// TIA Portal V15.1 export
// export: Created 2024-06-21T08:41:13.6587358Z, ExportSetting WithDefaults, DisplayName Totally Integrated Automation Portal, DisplayVersion V15.1 Update 5, DisplayName TIA Portal Openness, DisplayVersion V15.1 Update 5, DisplayName SINAMICS Startdrive Advanced, DisplayVersion V15.1, DisplayName G130, G150, S120, S150, SINAMICS MV, S210, DisplayVersion V15.1, DisplayName G110M, G120, G120C, G120D, G120P, DisplayVersion V15.1, DisplayName STEP 7 Professional, DisplayVersion V15.1 Update 5, DisplayName STEP 7 Safety, DisplayVersion V15.1, DisplayName WinCC Professional, DisplayVersion V15.1 Update 5, DisplayName SIMATIC Visualization Architect, DisplayVersion V15.1
FUNCTION_BLOCK "LGBLightCurtain"   // FB6634, FBD
TITLE = LGBLightCurtain
{ S7_Optimized_Access := 'FALSE' }
VERSION : 0.1
// ============================================================================
// This module is generates an alarm regarding a light curtain. The module manages also the bypass key and the pollution alarm.
// The light curtain alarm is reset by means of the AlarmResetPB signal.
// 
// This module generates also a word containing all necessary information for HMI 
// Icon animation, and a word with all information for HMI safety module diagnostic screen. 
// ============================================================================
// stored: AutoNumber false, IsIECCheckEnabled false, SetENOAutomatically False, UDAEnableTagReadback false
   VAR_INPUT
      I_LightCurtain { ExternalAccessible := 'False'; ExternalVisible := 'False'; ExternalWritable := 'False'} : Bool;   // Input safety (normally closed) / Input safety alarm (normally closed)
      I_Polluted { ExternalAccessible := 'False'; ExternalVisible := 'False'; ExternalWritable := 'False'} : Bool;   // Light curtain is polluted / Input safety alarm (normally closed)
      I_MutingAlarm { ExternalAccessible := 'False'; ExternalVisible := 'False'; ExternalWritable := 'False'} : Bool;   // Muting alarm from safety FB "MUT_P"
      I_OkToReset { ExternalAccessible := 'False'; ExternalVisible := 'False'; ExternalWritable := 'False'} : Bool;   // Ok to Reset Light curtain
      I_BypassKey { ExternalAccessible := 'False'; ExternalVisible := 'False'; ExternalWritable := 'False'} : Bool;   // Light curtain override key is turned / Input safety alarm (normally closed)
      I_AlarmClassLightCurtain { ExternalAccessible := 'False'; ExternalVisible := 'False'; ExternalWritable := 'False'} : Char;   // Alarm class -> A - B - C - D or E
      I_AlarmClassMuting { ExternalAccessible := 'False'; ExternalVisible := 'False'; ExternalWritable := 'False'} : Char;   // Alarm class -> A - B - C - D or E
      I_EnableAlarm { ExternalAccessible := 'False'; ExternalVisible := 'False'; ExternalWritable := 'False'} : Bool := TRUE;   // Enable alarm from upper level
      I_AlarmResetPB { ExternalAccessible := 'False'; ExternalVisible := 'False'; ExternalWritable := 'False'} : Bool;   // Alarm reset pushbutton is activated
      I_ResetAlarmPolluted { ExternalAccessible := 'False'; ExternalVisible := 'False'; ExternalWritable := 'False'} : Bool;   // Reset polluted alarm / Alarm reset pushbutton is activated
      I_SafetyCard_PASS_OUT { ExternalAccessible := 'False'; ExternalVisible := 'False'; ExternalWritable := 'False'} : Bool;   // Automatically generated DB from F-Modul (F-Peripherie DB)
      I_SafetyCard_ACK_REQ { ExternalAccessible := 'False'; ExternalVisible := 'False'; ExternalWritable := 'False'} : Bool;   // Automatically generated DB from F-Modul (F-Peripherie DB)
      I_SafetyCard_DIAG { ExternalAccessible := 'False'; ExternalVisible := 'False'; ExternalWritable := 'False'} : Byte;   // Automatically generated DB from F-Modul (F-Peripherie DB)
      I_SafetyCardHWSub { ExternalAccessible := 'False'; ExternalVisible := 'False'; ExternalWritable := 'False'} : HW_SUBMODULE;   // Safety I/O connection hardware
      I_ChannelNr { ExternalAccessible := 'False'; ExternalVisible := 'False'; ExternalWritable := 'False'} : Int;   // Used Channel Nr (Value : 0, 1, 2, 3)
      C_DisableQBadCh { ExternalAccessible := 'False'; ExternalVisible := 'False'; ExternalWritable := 'False'} : Bool;   // Passivation Channel (QbadCh1) / Disable QBad Channel
      C_DisablePollutedAlarm { ExternalAccessible := 'False'; ExternalVisible := 'False'; ExternalWritable := 'False'} : Bool;   // Disable Polluted Alarm
   END_VAR
   VAR_OUTPUT
      O_AlarmABCondition { ExternalAccessible := 'False'; ExternalVisible := 'False'; ExternalWritable := 'False'} : Bool;   // Alarm AB condition
      O_AlarmA { ExternalAccessible := 'False'; ExternalVisible := 'False'; ExternalWritable := 'False'} : Bool;   // Alarm A
      O_AlarmB { ExternalAccessible := 'False'; ExternalVisible := 'False'; ExternalWritable := 'False'} : Bool;   // Alarm B
      O_AlarmC { ExternalAccessible := 'False'; ExternalVisible := 'False'; ExternalWritable := 'False'} : Bool;   // Alarm C
      O_AlarmD { ExternalAccessible := 'False'; ExternalVisible := 'False'; ExternalWritable := 'False'} : Bool;   // Alarm D
      H_IAnim { ExternalAccessible := 'False'; ExternalVisible := 'False'; ExternalWritable := 'False'} : DWord;   // Icon Animation
      H_AlarmWord { ExternalAccessible := 'False'; ExternalVisible := 'False'; ExternalWritable := 'False'} : DWord;   // Alarm Word
   END_VAR
   VAR DB_SPECIFIC
      H_Out : Struct   // HMI
         Anim : Word;   // HMI Animation of the object
         DBnr : Int;   // HMI Animation DB number
      END_STRUCT;
      AlarmClassLightCurtain_A { ExternalAccessible := 'False'; ExternalVisible := 'False'; ExternalWritable := 'False'} : Bool;   // The alarm is from alarm class A / The alarm is from alarm Light Curtain class A
      AlarmClassLightCurtain_B { ExternalAccessible := 'False'; ExternalVisible := 'False'; ExternalWritable := 'False'} : Bool;   // The alarm is from alarm class B / The alarm is from alarm Light Curtain class B
      AlarmClassLightCurtain_C { ExternalAccessible := 'False'; ExternalVisible := 'False'; ExternalWritable := 'False'} : Bool;   // The alarm is from alarm class C / The alarm is from alarm Light Curtain class C
      AlarmClassLightCurtain_D { ExternalAccessible := 'False'; ExternalVisible := 'False'; ExternalWritable := 'False'} : Bool;   // The alarm is from alarm class D / The alarm is from alarm Light Curtain class D
      AlarmClassMuting_A { ExternalAccessible := 'False'; ExternalVisible := 'False'; ExternalWritable := 'False'} : Bool;   // The alarm is from alarm class A / The alarm is from alarm Muting class A
      AlarmClassMuting_B { ExternalAccessible := 'False'; ExternalVisible := 'False'; ExternalWritable := 'False'} : Bool;   // The alarm is from alarm class B / The alarm is from alarm Muting class B
      AlarmClassMuting_C { ExternalAccessible := 'False'; ExternalVisible := 'False'; ExternalWritable := 'False'} : Bool;   // The alarm is from alarm class C / The alarm is from alarm Muting class C
      AlarmClassMuting_D { ExternalAccessible := 'False'; ExternalVisible := 'False'; ExternalWritable := 'False'} : Bool;   // The alarm is from alarm class D / The alarm is from alarm Muting class D
      Alarm { ExternalAccessible := 'False'; ExternalVisible := 'False'; ExternalWritable := 'False'} : Bool;   // Alarm
      AA_LightCurtainAlarm { ExternalAccessible := 'False'; ExternalVisible := 'False'; ExternalWritable := 'False'} : Bool;   // Alarm of the light curtain / Alarm
      AB_LightCurtainAlarm { ExternalAccessible := 'False'; ExternalVisible := 'False'; ExternalWritable := 'False'} : Bool;   // Alarm of the light curtain / Alarm
      AC_LightCurtainAlarm { ExternalAccessible := 'False'; ExternalVisible := 'False'; ExternalWritable := 'False'} : Bool;   // Alarm of the light curtain / Alarm
      AD_LightCurtainAlarm { ExternalAccessible := 'False'; ExternalVisible := 'False'; ExternalWritable := 'False'} : Bool;   // Alarm of the light curtain / Alarm
      AA_MutingAlarm { ExternalAccessible := 'False'; ExternalVisible := 'False'; ExternalWritable := 'False'} : Bool;   // Muting is not ok
      AB_MutingAlarm { ExternalAccessible := 'False'; ExternalVisible := 'False'; ExternalWritable := 'False'} : Bool;   // Muting is not ok
      AC_MutingAlarm { ExternalAccessible := 'False'; ExternalVisible := 'False'; ExternalWritable := 'False'} : Bool;   // Muting is not ok
      AD_MutingAlarm { ExternalAccessible := 'False'; ExternalVisible := 'False'; ExternalWritable := 'False'} : Bool;   // Muting is not ok
      AC_Polluted { ExternalAccessible := 'False'; ExternalVisible := 'False'; ExternalWritable := 'False'} : Bool;   // Light curtain is polluted / Alarm
      AC_Bypass { ExternalAccessible := 'False'; ExternalVisible := 'False'; ExternalWritable := 'False'} : Bool;   // Bypass key is activated / Alarm
      QbadCh1 { ExternalAccessible := 'False'; ExternalVisible := 'False'; ExternalWritable := 'False'} : Bool;   // Passivation first Channel
      Ack_Req { ExternalAccessible := 'False'; ExternalVisible := 'False'; ExternalWritable := 'False'} : Bool;   // Acknowledgement request
      Timeout_F_I_O { ExternalAccessible := 'False'; ExternalVisible := 'False'; ExternalWritable := 'False'} : Bool;   // Timeout detected by F-I/O
      ChannelFault_F_I_O { ExternalAccessible := 'False'; ExternalVisible := 'False'; ExternalWritable := 'False'} : Bool;   // F-I/O fault or channel fault detected by F-I/O
      CRCSeqError_F_I_O { ExternalAccessible := 'False'; ExternalVisible := 'False'; ExternalWritable := 'False'} : Bool;   // CRC error or sequence number error detected by F-I/O
      Timeout_F_Sys { ExternalAccessible := 'False'; ExternalVisible := 'False'; ExternalWritable := 'False'} : Bool;   // Timeout detected by F-System
      SeqError_F_Sys { ExternalAccessible := 'False'; ExternalVisible := 'False'; ExternalWritable := 'False'} : Bool;   // Sequence number error detected by F-system
      CRCError_F_Sys { ExternalAccessible := 'False'; ExternalVisible := 'False'; ExternalWritable := 'False'} : Bool;   // CRC error detected by F-system
      AlarmCond { ExternalAccessible := 'False'; ExternalVisible := 'False'; ExternalWritable := 'False'} : Bool;   // Alarm condition
      RetValueData { ExternalAccessible := 'False'; ExternalVisible := 'False'; ExternalWritable := 'False'} : Int;   // Status variable (SFC14)
      DBnr { ExternalAccessible := 'False'; ExternalVisible := 'False'; ExternalWritable := 'False'} : Int;   // HMI DB number
      AlarmABCondition { ExternalAccessible := 'False'; ExternalVisible := 'False'; ExternalWritable := 'False'} : Bool;   // Alarm AB Condition / Summation Alarm A
      AlarmA { ExternalAccessible := 'False'; ExternalVisible := 'False'; ExternalWritable := 'False'} : Bool;   // Summation Alarm A
      AlarmB { ExternalAccessible := 'False'; ExternalVisible := 'False'; ExternalWritable := 'False'} : Bool;   // Summation Alarm B
      AlarmC { ExternalAccessible := 'False'; ExternalVisible := 'False'; ExternalWritable := 'False'} : Bool;   // Summation Alarm C
      AlarmD { ExternalAccessible := 'False'; ExternalVisible := 'False'; ExternalWritable := 'False'} : Bool;   // Summation Alarm D
   END_VAR
   VAR_TEMP
      T_DataFromSafetyCard : Struct   // Temp structure : receive data's from Safety Card
         Byte0_Bit0_Spare : Bool;
         Byte0_Bit1_Spare : Bool;
         Byte0_Bit2_Spare : Bool;
         Byte0_Bit3_Spare : Bool;
         Byte0_Bit4_Spare : Bool;
         Byte0_Bit5_Spare : Bool;
         Byte0_Bit6_Spare : Bool;
         Byte0_Bit7_Spare : Bool;
         Byte1_Bit0_QBadCh0 : Bool;
         Byte1_Bit1_QBadCh1 : Bool;
         Byte1_Bit2_QBadCh2 : Bool;
         Byte1_Bit3_QBadCh3 : Bool;
         Byte1_Bit4_QBadCh4 : Bool;
         Byte1_Bit5_QBadCh5 : Bool;
         Byte1_Bit6_QBadCh6 : Bool;
         Byte1_Bit7_QBadCh7 : Bool;
         Byte2_bit0_Spare : Bool;
         Byte2_bit1_Spare : Bool;
         Byte2_bit2_Spare : Bool;
         Byte2_bit3_Spare : Bool;
         Byte2_bit4_Spare : Bool;
         Byte2_bit5_Spare : Bool;
         Byte2_bit6_Spare : Bool;
         Byte2_bit7_Spare : Bool;
         Byte3_Bit0_Spare : Bool;
         Byte3_Bit1_Spare : Bool;
         Byte3_Bit2_Spare : Bool;
         Byte3_Bit3_Spare : Bool;
         Byte3_Bit4_Spare : Bool;
         Byte3_Bit5_Spare : Bool;
         Byte3_Bit6_Spare : Bool;
         Byte3_Bit7_Spare : Bool;
         Byte4_bit0_Spare : Bool;
         Byte4_bit1_Spare : Bool;
         Byte4_bit2_Spare : Bool;
         Byte4_bit3_Spare : Bool;
         Byte4_bit4_Spare : Bool;
         Byte4_bit5_Spare : Bool;
         Byte4_bit6_Spare : Bool;
         Byte4_bit7_Spare : Bool;
         Byte5_bit0_Spare : Bool;
         Byte5_bit1_Spare : Bool;
         Byte5_bit2_Spare : Bool;
         Byte5_bit3_Spare : Bool;
         Byte5_bit4_Spare : Bool;
         Byte5_bit5_Spare : Bool;
         Byte5_bit6_Spare : Bool;
         Byte5_bit7_Spare : Bool;
      END_STRUCT;
   END_VAR
   VAR_TEMP   // added for the SCL form of the ladder/FBD networks
      _w1 : Bool;
   END_VAR
BEGIN

NETWORK
TITLE = **** 1 - Inputs **** DB number
// DB number
      L     DINO;
      T     #DBnr;

NETWORK
TITLE = **** 1 - Inputs **** Alarm class / **** 1 - Inputs **** Alarm class Light Curtain
// Alarm class
// Alarm class = D
      L     #I_AlarmClassLightCurtain;
      L     'D';
      ==I;
      =     #AlarmClassLightCurtain_D;

// Alarm class = C
      L     #I_AlarmClassLightCurtain;
      L     'C';
      ==I;
      =     #AlarmClassLightCurtain_C;

// Alarm class = B
      L     #I_AlarmClassLightCurtain;
      L     'B';
      ==I;
      =     #AlarmClassLightCurtain_B;

// Alarm class = A
      AN    #AlarmClassLightCurtain_B;
      AN    #AlarmClassLightCurtain_C;
      AN    #AlarmClassLightCurtain_D;
      =     #AlarmClassLightCurtain_A;


NETWORK
TITLE = **** 1 - Inputs **** Alarm class / **** 1 - Inputs **** Alarm class Muting
// Alarm class
// Alarm class = D
      L     #I_AlarmClassMuting;
      L     'D';
      ==I;
      =     #AlarmClassMuting_D;

// Alarm class = C
      L     #I_AlarmClassMuting;
      L     'C';
      ==I;
      =     #AlarmClassMuting_C;

// Alarm class = B
      L     #I_AlarmClassMuting;
      L     'B';
      ==I;
      =     #AlarmClassMuting_B;

// Alarm class = A
      AN    #AlarmClassMuting_B;
      AN    #AlarmClassMuting_C;
      AN    #AlarmClassMuting_D;
      =     #AlarmClassMuting_A;


REGION Network 4: **** 1 - Inputs **** Safety I/O connection hardware
   // Safety I/O connection hardware
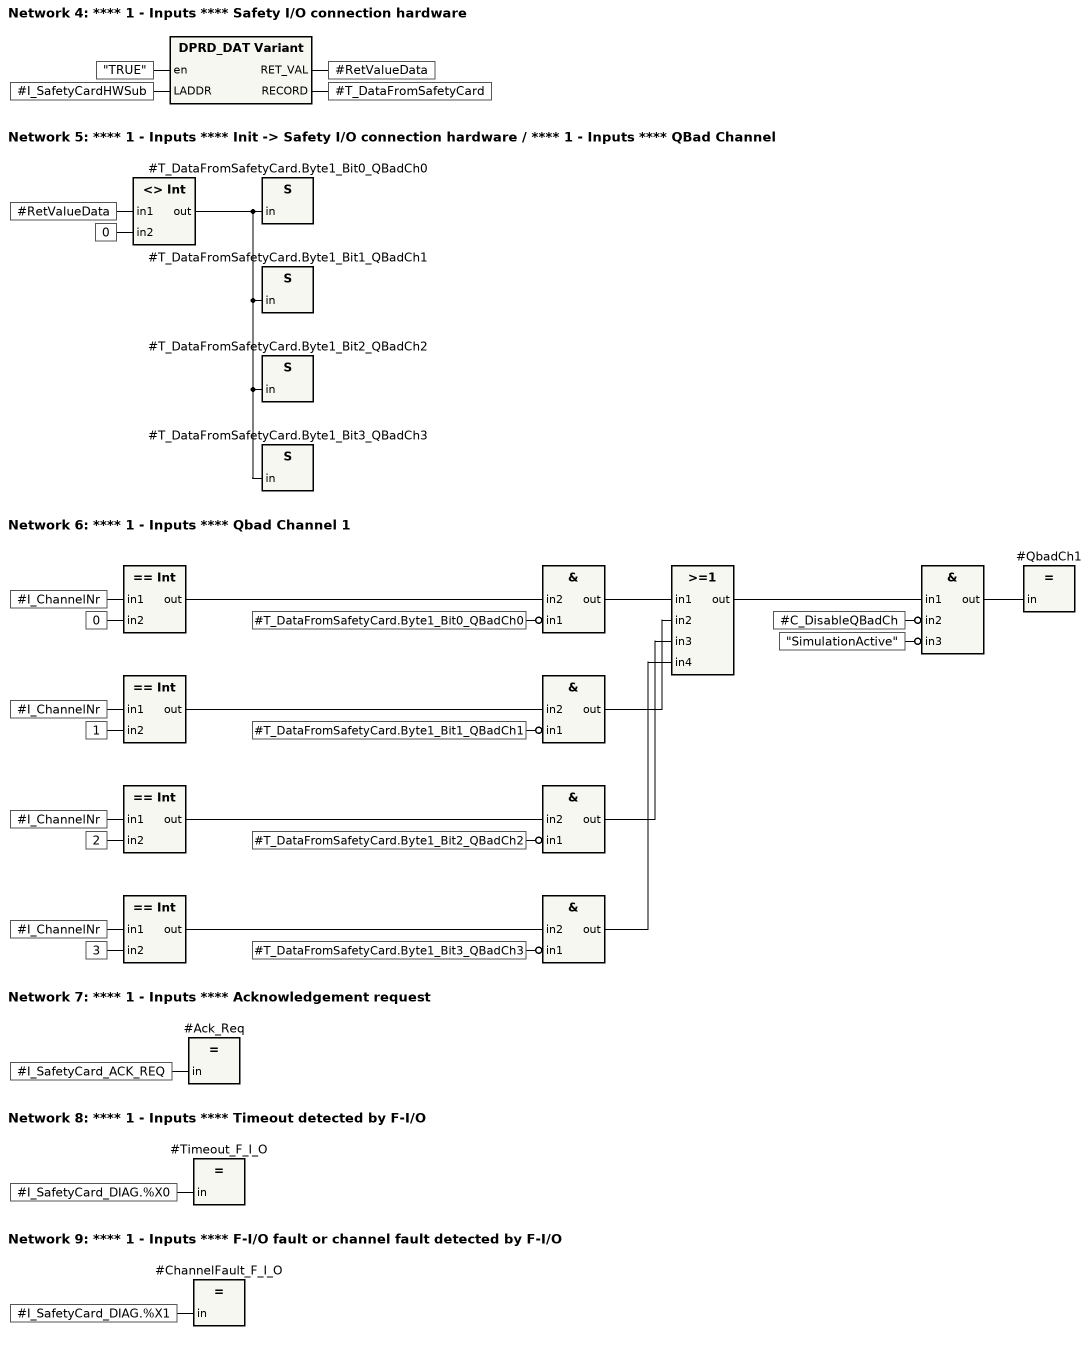
   IF "TRUE" THEN
       #RetValueData := DPRD_DAT(LADDR := #I_SafetyCardHWSub, RECORD => #T_DataFromSafetyCard);
   END_IF;
END_REGION

REGION Network 5: **** 1 - Inputs **** Init -> Safety I/O connection hardware / **** 1 - Inputs **** QBad Channel
   // Init -> Safety I/O connection hardware
   IF #RetValueData <> 0 THEN
       #T_DataFromSafetyCard.Byte1_Bit0_QBadCh0 := TRUE;
       #T_DataFromSafetyCard.Byte1_Bit1_QBadCh1 := TRUE;
       #T_DataFromSafetyCard.Byte1_Bit2_QBadCh2 := TRUE;
       #T_DataFromSafetyCard.Byte1_Bit3_QBadCh3 := TRUE;
   END_IF;
END_REGION

REGION Network 6: **** 1 - Inputs **** Qbad Channel 1
   // Qbad Channel 1
   #QbadCh1 := (((#I_ChannelNr = 0) AND NOT #T_DataFromSafetyCard.Byte1_Bit0_QBadCh0) OR ((#I_ChannelNr = 1) AND NOT #T_DataFromSafetyCard.Byte1_Bit1_QBadCh1) OR ((#I_ChannelNr = 2) AND NOT #T_DataFromSafetyCard.Byte1_Bit2_QBadCh2) OR ((#I_ChannelNr = 3) AND NOT #T_DataFromSafetyCard.Byte1_Bit3_QBadCh3)) AND NOT #C_DisableQBadCh AND NOT "SimulationActive";
END_REGION

REGION Network 7: **** 1 - Inputs **** Acknowledgement request
   // Acknowledgement request
   #Ack_Req := #I_SafetyCard_ACK_REQ;
END_REGION

REGION Network 8: **** 1 - Inputs **** Timeout detected by F-I/O
   // Timeout detected by F-I/O
   #Timeout_F_I_O := #I_SafetyCard_DIAG.%X0;
END_REGION

REGION Network 9: **** 1 - Inputs **** F-I/O fault or channel fault detected by F-I/O
   // F-I/O fault or channel fault detected by F-I/O
   #ChannelFault_F_I_O := #I_SafetyCard_DIAG.%X1;
END_REGION

REGION Network 10: **** 1 - Inputs **** CRC error or sequence number error detected by F-I/O
   // CRC error or sequence number error detected by F-I/O
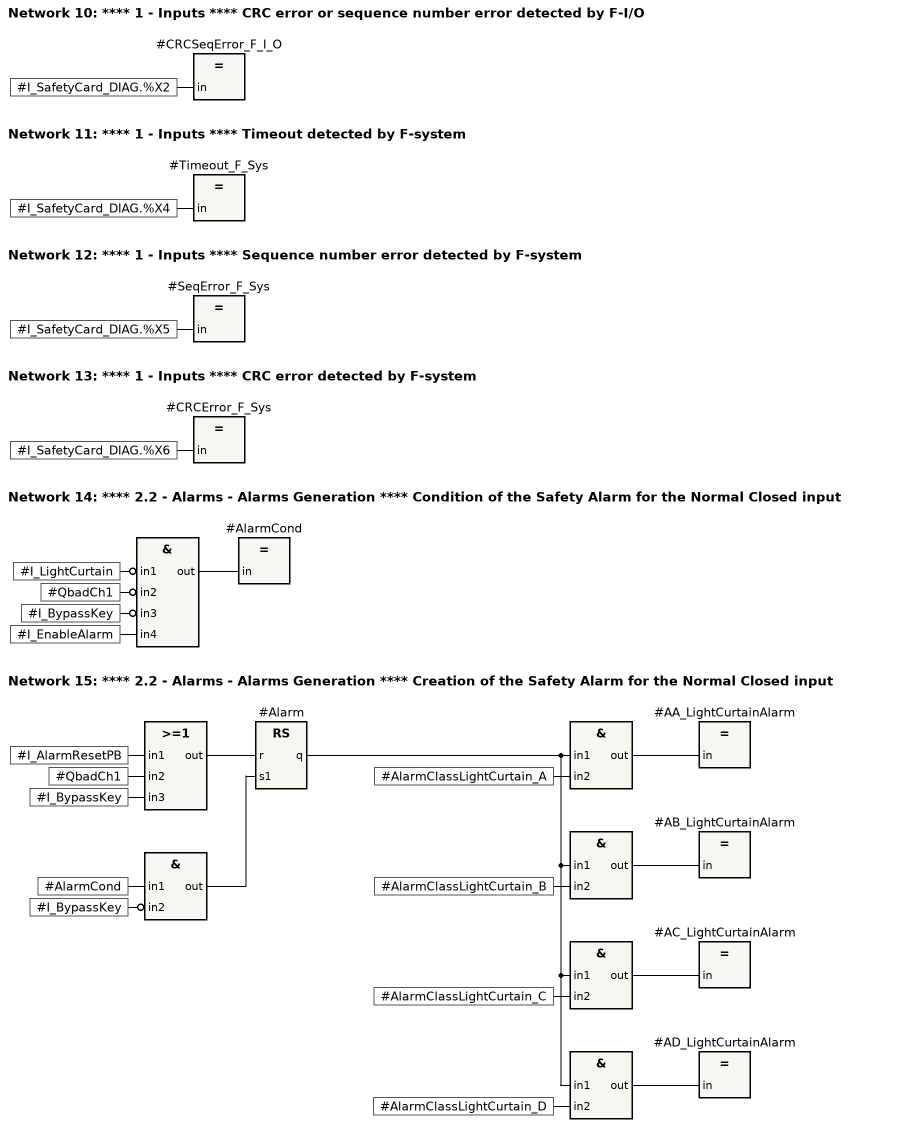
   #CRCSeqError_F_I_O := #I_SafetyCard_DIAG.%X2;
END_REGION

REGION Network 11: **** 1 - Inputs **** Timeout detected by F-system
   // Timeout detected by F-system
   #Timeout_F_Sys := #I_SafetyCard_DIAG.%X4;
END_REGION

REGION Network 12: **** 1 - Inputs **** Sequence number error detected by F-system
   // Sequence number error detected by F-system
   #SeqError_F_Sys := #I_SafetyCard_DIAG.%X5;
END_REGION

REGION Network 13: **** 1 - Inputs **** CRC error detected by F-system
   // CRC error detected by F-system
   #CRCError_F_Sys := #I_SafetyCard_DIAG.%X6;
END_REGION

REGION Network 14: **** 2.2 - Alarms - Alarms Generation **** Condition of the Safety Alarm for the Normal Closed input
   // Condition of the Safety Alarm for the Normal Closed input
   #AlarmCond := NOT #I_LightCurtain AND NOT #QbadCh1 AND NOT #I_BypassKey AND #I_EnableAlarm;
END_REGION

REGION Network 15: **** 2.2 - Alarms - Alarms Generation **** Creation of the Safety Alarm for the Normal Closed input
   // Creation of the Safety Alarm for the Normal Closed input
   IF #I_AlarmResetPB OR #QbadCh1 OR #I_BypassKey THEN
       #Alarm := FALSE;   // RS flip-flop
   END_IF;
   IF #AlarmCond AND NOT #I_BypassKey THEN #Alarm := TRUE; END_IF;
   #AA_LightCurtainAlarm := #Alarm AND #AlarmClassLightCurtain_A;
   #AB_LightCurtainAlarm := #Alarm AND #AlarmClassLightCurtain_B;
   #AC_LightCurtainAlarm := #Alarm AND #AlarmClassLightCurtain_C;
   #AD_LightCurtainAlarm := #Alarm AND #AlarmClassLightCurtain_D;
END_REGION

REGION Network 16: **** 2.2 - Alarms - Alarms Generation **** Muting is not ok
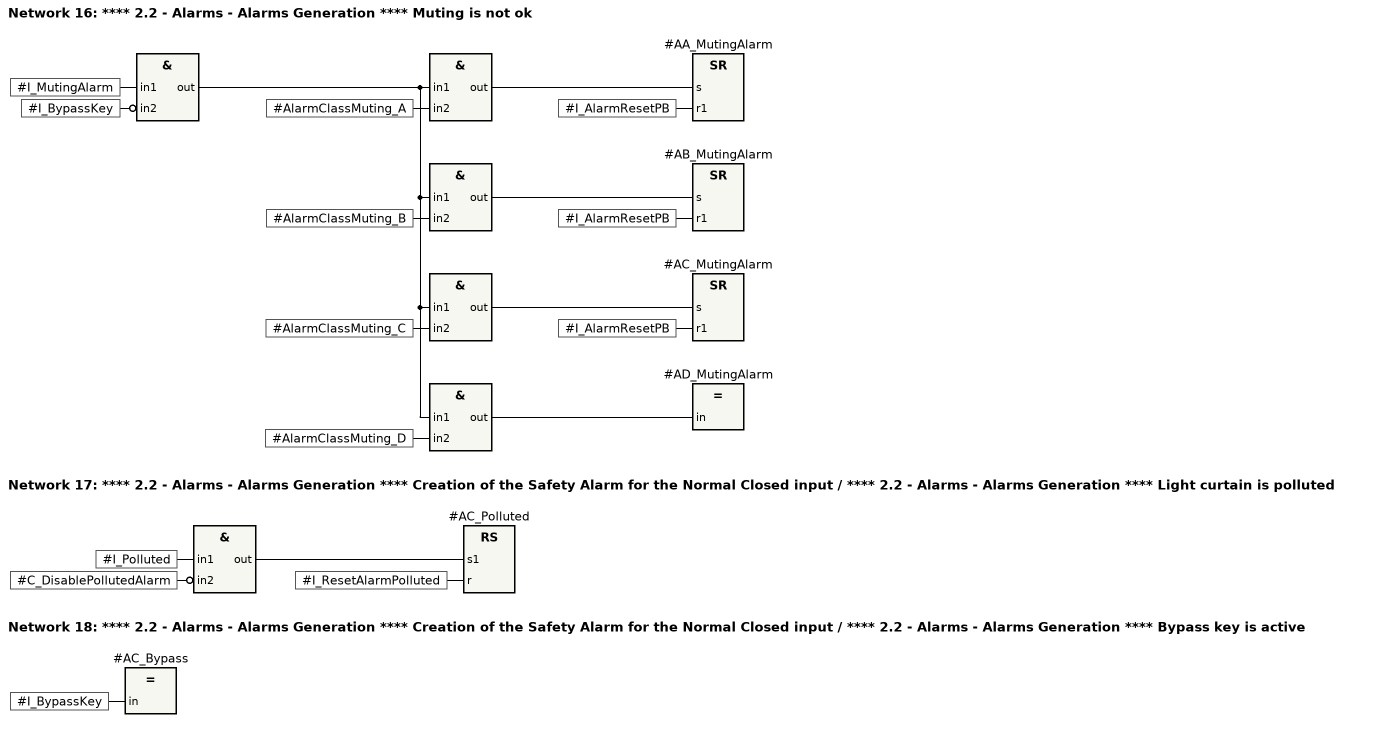
   #_w1 := #I_MutingAlarm AND NOT #I_BypassKey;
   IF #_w1 AND #AlarmClassMuting_A THEN
       #AA_MutingAlarm := TRUE;   // SR flip-flop
   END_IF;
   IF #I_AlarmResetPB THEN #AA_MutingAlarm := FALSE; END_IF;
   IF #_w1 AND #AlarmClassMuting_B THEN
       #AB_MutingAlarm := TRUE;   // SR flip-flop
   END_IF;
   IF #I_AlarmResetPB THEN #AB_MutingAlarm := FALSE; END_IF;
   IF #_w1 AND #AlarmClassMuting_C THEN
       #AC_MutingAlarm := TRUE;   // SR flip-flop
   END_IF;
   IF #I_AlarmResetPB THEN #AC_MutingAlarm := FALSE; END_IF;
   #AD_MutingAlarm := #_w1 AND #AlarmClassMuting_D;
END_REGION

REGION Network 17: **** 2.2 - Alarms - Alarms Generation **** Creation of the Safety Alarm for the Normal Closed input / **** 2.2 - Alarms - Alarms Generation **** Light curtain is polluted
   // Creation of the Safety Alarm for the Normal Closed input / Light curtain is polluted
   IF #I_ResetAlarmPolluted THEN
       #AC_Polluted := FALSE;   // RS flip-flop
   END_IF;
   IF #I_Polluted AND NOT #C_DisablePollutedAlarm THEN #AC_Polluted := TRUE; END_IF;
END_REGION

REGION Network 18: **** 2.2 - Alarms - Alarms Generation **** Creation of the Safety Alarm for the Normal Closed input / **** 2.2 - Alarms - Alarms Generation **** Bypass key is active
   // Creation of the Safety Alarm for the Normal Closed input / Bypass key is active
   #AC_Bypass := #I_BypassKey;
END_REGION

REGION Network 19: **** 4.6 - Machine Status - Indications **** Icon Animation
   // Icon Animation
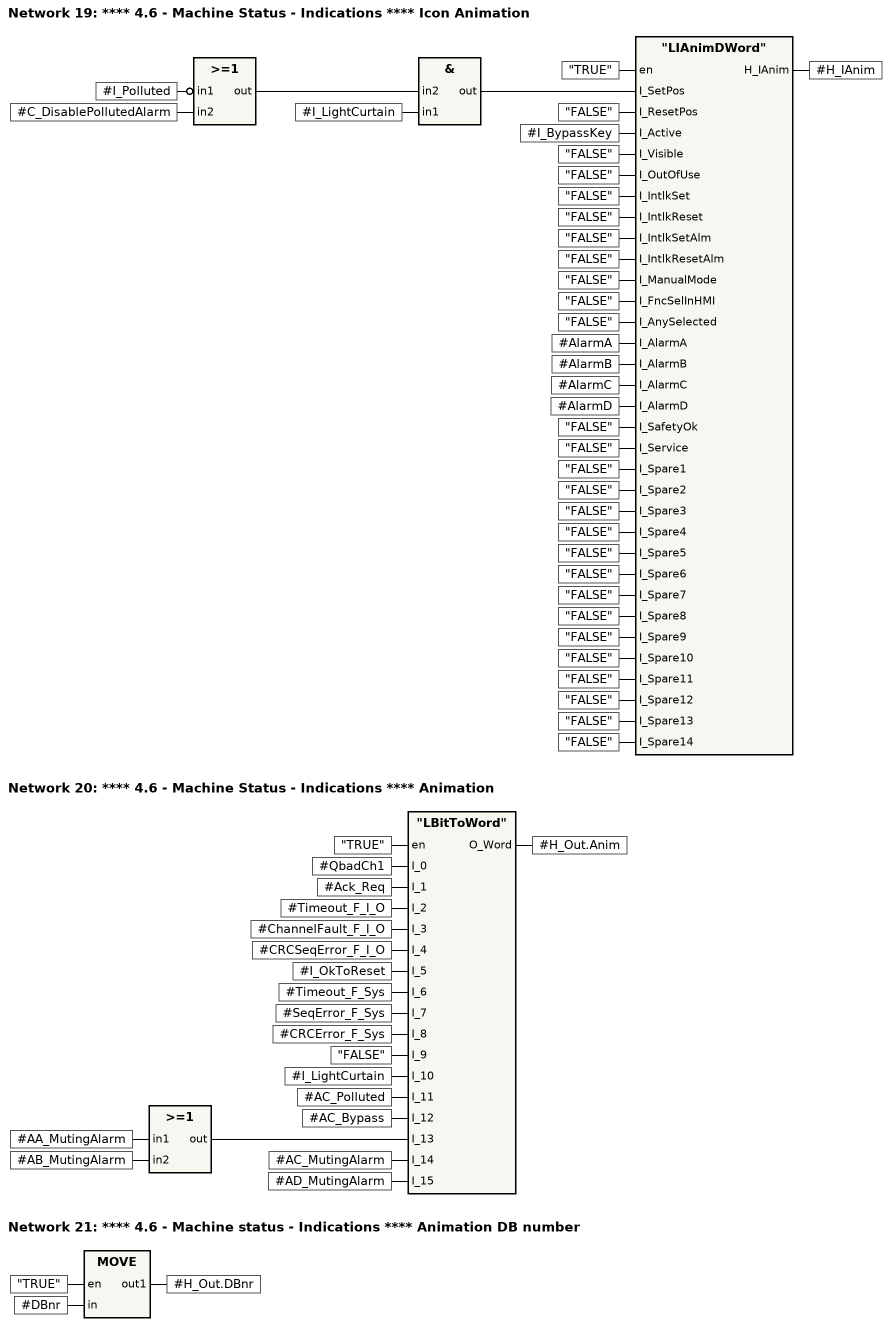
   IF "TRUE" THEN
       "LIAnimDWord"(I_SetPos := (NOT #I_Polluted OR #C_DisablePollutedAlarm) AND #I_LightCurtain,
                     I_ResetPos := "FALSE",
                     I_Active := #I_BypassKey,
                     I_Visible := "FALSE",
                     I_OutOfUse := "FALSE",
                     I_IntlkSet := "FALSE",
                     I_IntlkReset := "FALSE",
                     I_IntlkSetAlm := "FALSE",
                     I_IntlkResetAlm := "FALSE",
                     I_ManualMode := "FALSE",
                     I_FncSelInHMI := "FALSE",
                     I_AnySelected := "FALSE",
                     I_AlarmA := #AlarmA,
                     I_AlarmB := #AlarmB,
                     I_AlarmC := #AlarmC,
                     I_AlarmD := #AlarmD,
                     I_SafetyOk := "FALSE",
                     I_Service := "FALSE",
                     I_Spare1 := "FALSE",
                     I_Spare2 := "FALSE",
                     I_Spare3 := "FALSE",
                     I_Spare4 := "FALSE",
                     I_Spare5 := "FALSE",
                     I_Spare6 := "FALSE",
                     I_Spare7 := "FALSE",
                     I_Spare8 := "FALSE",
                     I_Spare9 := "FALSE",
                     I_Spare10 := "FALSE",
                     I_Spare11 := "FALSE",
                     I_Spare12 := "FALSE",
                     I_Spare13 := "FALSE",
                     I_Spare14 := "FALSE",
                     H_IAnim => #H_IAnim);
   END_IF;
END_REGION

REGION Network 20: **** 4.6 - Machine Status - Indications **** Animation
   // Animation
   IF "TRUE" THEN
       "LBitToWord"(I_0 := #QbadCh1,
                    I_1 := #Ack_Req,
                    I_2 := #Timeout_F_I_O,
                    I_3 := #ChannelFault_F_I_O,
                    I_4 := #CRCSeqError_F_I_O,
                    I_5 := #I_OkToReset,
                    I_6 := #Timeout_F_Sys,
                    I_7 := #SeqError_F_Sys,
                    I_8 := #CRCError_F_Sys,
                    I_9 := "FALSE",
                    I_10 := #I_LightCurtain,
                    I_11 := #AC_Polluted,
                    I_12 := #AC_Bypass,
                    I_13 := #AA_MutingAlarm OR #AB_MutingAlarm,
                    I_14 := #AC_MutingAlarm,
                    I_15 := #AD_MutingAlarm,
                    O_Word => #H_Out.Anim);
   END_IF;
END_REGION

REGION Network 21: **** 4.6 - Machine status - Indications **** Animation DB number
   // Animation DB number
   IF "TRUE" THEN #H_Out.DBnr := #DBnr; END_IF;
END_REGION

REGION Network 22: **** 8 - Outputs **** Output of the alarm AB condition / **** 9 - Alarm Summary **** Alarm AB condition
   // Alarm AB condition
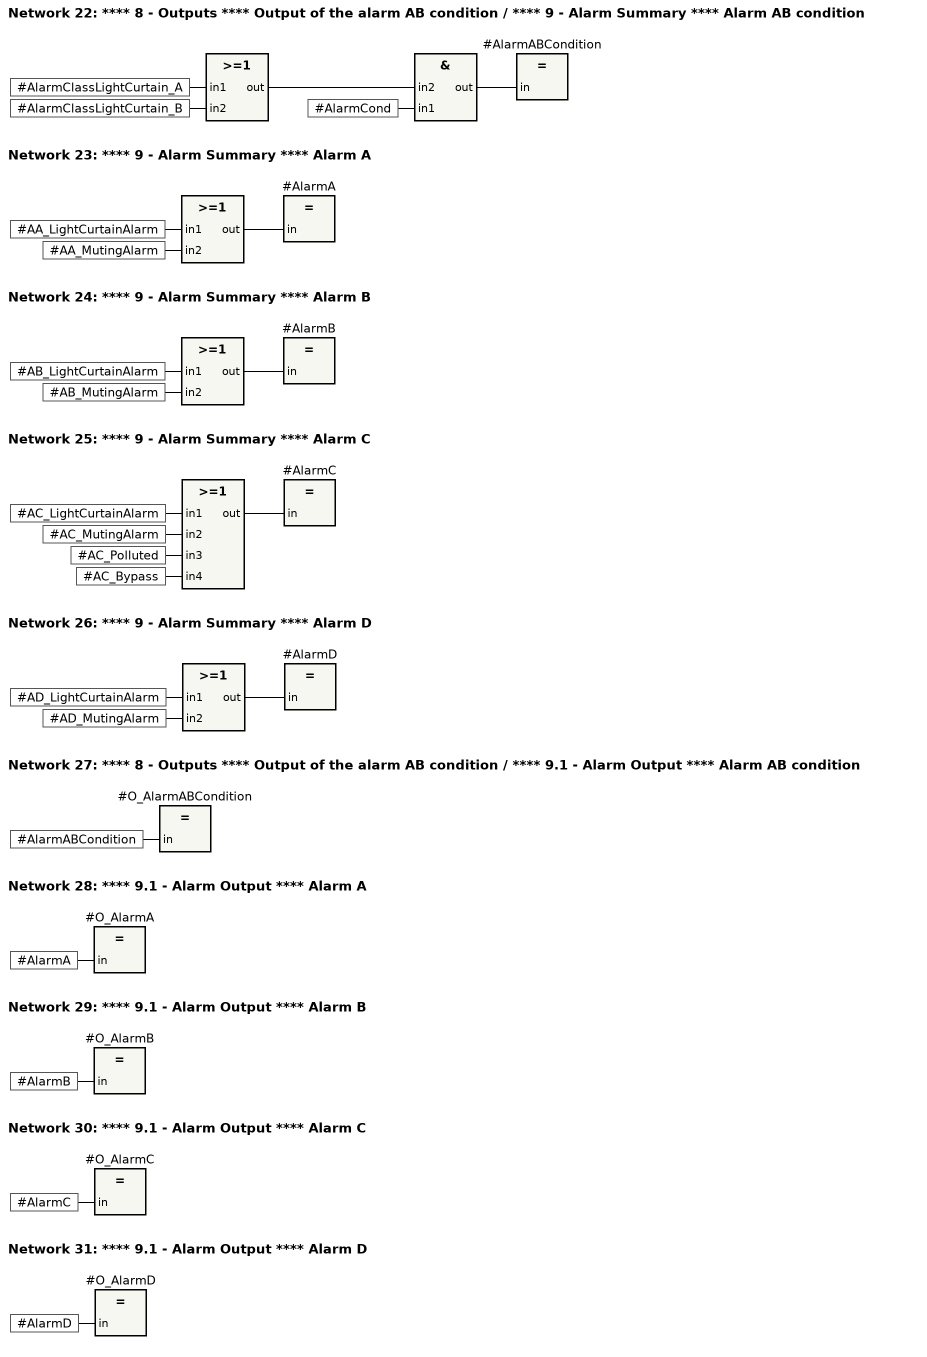
   #AlarmABCondition := (#AlarmClassLightCurtain_A OR #AlarmClassLightCurtain_B) AND #AlarmCond;
END_REGION

REGION Network 23: **** 9 - Alarm Summary **** Alarm A
   // Alarm A
   #AlarmA := #AA_LightCurtainAlarm OR #AA_MutingAlarm;
END_REGION

REGION Network 24: **** 9 - Alarm Summary **** Alarm B
   // Alarm B
   #AlarmB := #AB_LightCurtainAlarm OR #AB_MutingAlarm;
END_REGION

REGION Network 25: **** 9 - Alarm Summary **** Alarm C
   // Alarm C
   #AlarmC := #AC_LightCurtainAlarm OR #AC_MutingAlarm OR #AC_Polluted OR #AC_Bypass;
END_REGION

REGION Network 26: **** 9 - Alarm Summary **** Alarm D
   // Alarm D
   #AlarmD := #AD_LightCurtainAlarm OR #AD_MutingAlarm;
END_REGION

REGION Network 27: **** 8 - Outputs **** Output of the alarm AB condition / **** 9.1 - Alarm Output **** Alarm AB condition
   // Alarm AB condition
   #O_AlarmABCondition := #AlarmABCondition;
END_REGION

REGION Network 28: **** 9.1 - Alarm Output **** Alarm A
   // Alarm A
   #O_AlarmA := #AlarmA;
END_REGION

REGION Network 29: **** 9.1 - Alarm Output **** Alarm B
   // Alarm B
   #O_AlarmB := #AlarmB;
END_REGION

REGION Network 30: **** 9.1 - Alarm Output **** Alarm C
   // Alarm C
   #O_AlarmC := #AlarmC;
END_REGION

REGION Network 31: **** 9.1 - Alarm Output **** Alarm D
   // Alarm D
   #O_AlarmD := #AlarmD;
END_REGION

REGION Network 32: **** 9.2 - Alarm DWord**** Alarm To DWord
   // Alarm Word
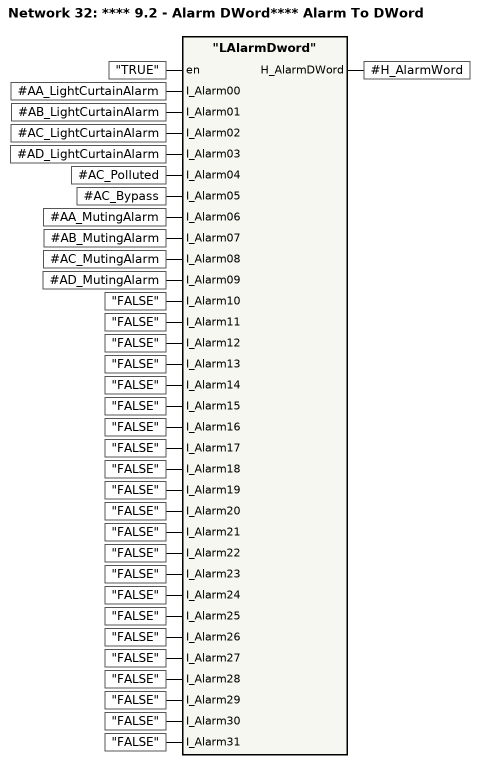
   IF "TRUE" THEN
       "LAlarmDword"(I_Alarm00 := #AA_LightCurtainAlarm,
                     I_Alarm01 := #AB_LightCurtainAlarm,
                     I_Alarm02 := #AC_LightCurtainAlarm,
                     I_Alarm03 := #AD_LightCurtainAlarm,
                     I_Alarm04 := #AC_Polluted,
                     I_Alarm05 := #AC_Bypass,
                     I_Alarm06 := #AA_MutingAlarm,
                     I_Alarm07 := #AB_MutingAlarm,
                     I_Alarm08 := #AC_MutingAlarm,
                     I_Alarm09 := #AD_MutingAlarm,
                     I_Alarm10 := "FALSE",
                     I_Alarm11 := "FALSE",
                     I_Alarm12 := "FALSE",
                     I_Alarm13 := "FALSE",
                     I_Alarm14 := "FALSE",
                     I_Alarm15 := "FALSE",
                     I_Alarm16 := "FALSE",
                     I_Alarm17 := "FALSE",
                     I_Alarm18 := "FALSE",
                     I_Alarm19 := "FALSE",
                     I_Alarm20 := "FALSE",
                     I_Alarm21 := "FALSE",
                     I_Alarm22 := "FALSE",
                     I_Alarm23 := "FALSE",
                     I_Alarm24 := "FALSE",
                     I_Alarm25 := "FALSE",
                     I_Alarm26 := "FALSE",
                     I_Alarm27 := "FALSE",
                     I_Alarm28 := "FALSE",
                     I_Alarm29 := "FALSE",
                     I_Alarm30 := "FALSE",
                     I_Alarm31 := "FALSE",
                     H_AlarmDWord => #H_AlarmWord);
   END_IF;
END_REGION
END_FUNCTION_BLOCK
